Fanuc KAREL source: kb00171.KL

-- PROVISIONAL review KL for V940-1; original PC SHA256 d47685e47284b79da407e552f7b7a9bc65a128b949643f834f3cbbfe70ff4f78
-- Incomplete behavior may be omitted. Consult companion uncertainty JSON. Do not deploy.
PROGRAM KB00171
%NOLOCKGROUP
BEGIN
  -- V9_ZERO_TABLE_METADATA_HINT layout=0002_ascii; no indexed target words; source/name/runtime held
  -- UNRESOLVED_PC offsets 5-12; opcodes 9D,23
  -- UNRESOLVED_PC offsets 17-24; opcodes 9D,23
  -- UNRESOLVED_PC offsets 29-36; opcodes 9D,23
  -- UNRESOLVED_PC offsets 41-69; opcodes 27,22,22,22,31,23
  -- UNRESOLVED_PC offsets 74-78; opcodes 7F
END KB00171
